VAR_GLOBAL
	Tri1_Mot_Fw AT %Q* : BOOL; 
	Tri1_Mot_Bw AT %Q* : BOOL; 
	Cmp1_Mot_Fw AT %Q* : BOOL; 
	Cmp1_Mot_Bw AT %Q* : BOOL; 
	Piv1_Mot_Fw AT %Q* : BOOL; 
	Piv1_Mot_Bw AT %Q* : BOOL; 
	Tri2_Mot_Fw AT %Q* : BOOL; 
	Tri2_Mot_Bw AT %Q* : BOOL; 
	Tri3_Mot_Fw AT %Q* : BOOL; 
	Tri3_Mot_Bw AT %Q* : BOOL; 
	Gui1_Mot_Fw AT %Q* : BOOL; 
	Gui1_Mot_Bw AT %Q* : BOOL; 
	Gui2_Mot_Fw AT %Q* : BOOL; 
	Gui2_Mot_Bw AT %Q* : BOOL; 
	Cmp2_Mot_Fw AT %Q* : BOOL; 
	Cmp2_Mot_Bw AT %Q* : BOOL; 
	Tri4_Mot_Fw AT %Q* : BOOL; 
	Tri4_Mot_Bw AT %Q* : BOOL;  
END_VAR

(* stored: Version 1.1.0.1, ProductVersion 3.1.4026.11
   GVL GVL_LinearActuatorRelays: Id {5eab831f-9447-4481-a624-13723ab2af90} *)
